// LS Electric XG5000 project: 프로젝트최종 PLC
// PLC LSPLC
// module base 0 slot 0: 입출력 모듈:XBC-DR32H (DC 24V 입력, 릴레이 출력 32점)

PROGRAM NewProgram (task: 스캔 프로그램)

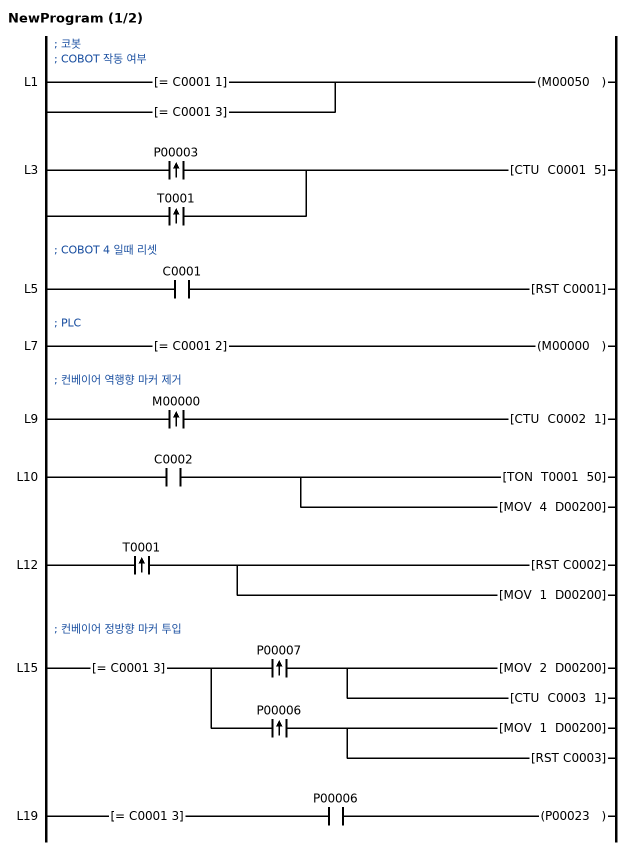
// 코봇
; L1
LOAD=     C0001 1
OR=       C0001 3
OUT       M00050
// output comment: COBOT 작동 여부
; L3
LOADP     P00003
ORP       T0001
CTU       C0001 5
; L5
LOAD      C0001
RST       C0001
// output comment: COBOT 4 일때 리셋
// PLC
; L7
LOAD=     C0001 2
OUT       M00000
// 컨베이어 역행향 마커 제거
; L9
LOADP     M00000
CTU       C0002 1
; L10
LOAD      C0002
TON       T0001 50
MOV       4 D00200
; L12
LOADP     T0001
RST       C0002
MOV       1 D00200
// 컨베이어 정방향 마커 투입
; L15
LOAD=     C0001 3
MPUSH
ANDP      P00007
MOV       2 D00200
CTU       C0003 1
MPOP
ANDP      P00006
MOV       1 D00200
RST       C0003
; L19
LOAD=     C0001 3
AND       P00006
OUT       P00023

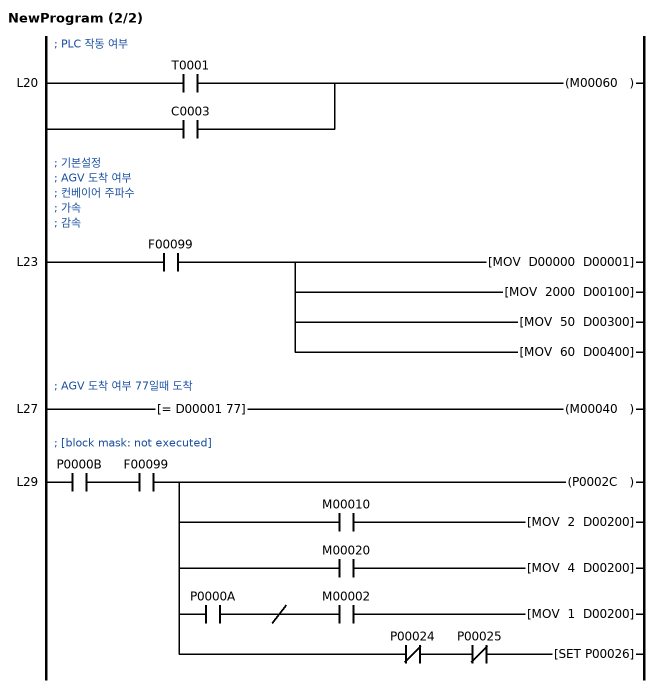
; L20
LOAD      T0001
OR        C0003
OUT       M00060
// output comment: PLC 작동 여부
// 기본설정
; L23
LOAD      F00099
MOV       D00000 D00001
MOV       2000 D00100
MOV       50 D00300
MOV       60 D00400
// output comment: AGV 도착 여부
// output comment: 컨베이어 주파수
// output comment: 가속
// output comment: 감속
; L27
LOAD=     D00001 77
OUT       M00040
// output comment: AGV 도착 여부 77일때 도착
; L29 (block mask: not executed)
LOAD      P0000B
AND       F00099
OUT       P0002C
MPUSH
AND       M00010
MOV       2 D00200
MLOAD
AND       M00020
MOV       4 D00200
MLOAD
AND       P0000A
NOT
AND       M00002
MOV       1 D00200
MPOP
AND NOT   P00024
AND NOT   P00025
SET       P00026